INTERFACE I_ChunkedResponseManager

METHOD PUBLIC HandleSuccess;
VAR_INPUT
	OriginalResponse : I_ServerResponse;
	SourceAddress : PVOID;
	SourceSize : UDINT;
END_VAR
END_METHOD

METHOD PUBLIC TryHandleIncomingRequest : BOOL
VAR_INPUT
	Request : I_Request;
	Response : I_ServerResponse;
END_VAR
END_METHOD

END_INTERFACE

(* stored: Version 1.1.0.1, ProductVersion 3.1.4024.12
   Itf I_ChunkedResponseManager: Id {62aad671-1eaf-4bad-a522-2f46caf7e50c}
   Method HandleSuccess: Id {90371fe9-8d96-473e-b2c5-d42ae6d2dbf7}
   Method TryHandleIncomingRequest: Id {879784c6-d759-44cb-9c64-5acc53f745df} *)
